{attribute 'qualified_only'}
{attribute 'strict'}
{attribute 'to_string'}
TYPE eModus :
(
	Off := 0,
	Auto := 1,
	Manual := 2
);
END_TYPE

(* stored: Version 1.1.0.1
   DUT eModus: Id {8a19fcfc-d24f-4f0f-8f76-7458174dc2b5} *)
